Staubli VAL3: save.pgx

public program save(string x_sName, num& x_nResult[])
begin
  // save it
  if isDefined(saveProg:pProg[x_sName]) and pEdit.iEvent.sType!=""
    saveProg:pProg[x_sName]=pEdit
  endIf
  x_nResult=saveProg:libSave()
end
